FUNCTION_BLOCK FB_PID_LIMI (* PID controller with limited frame for the integrator. *)
  (* Standard: 61499-2; Description: Rather than integrating the error over all vallues, the error is integrated over the last N values. Fixed-width time intervals are required for the input. *)
  (* Version 0.0, 2017-06-15, 4DIAC-IDE, 4DIAC-Consortium *)
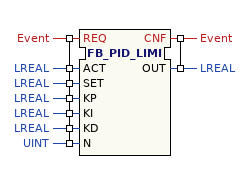
  EVENT_INPUT
    REQ WITH ACT, SET, KP, KI, KD, N; (* Normal Execution Request *)
  END_EVENT
  EVENT_OUTPUT
    CNF WITH OUT; (* Execution Confirmation *)
  END_EVENT
  VAR_INPUT
    ACT : LREAL; (* Actual value *)
    SET : LREAL; (* Set value *)
    KP : LREAL; (* Proportional coefficient *)
    KI : LREAL; (* Integral coefficient *)
    KD : LREAL; (* Derivative coefficient *)
    N : UINT := 1; (* Amount of values to look back for integral computation *)
  END_VAR
  VAR_OUTPUT
    OUT : LREAL; (* Output value = KP*(SET-ACT) + KI*INT_0_N(SET-ACT) + KD*DIFF(SET-ACT) *)
  END_VAR
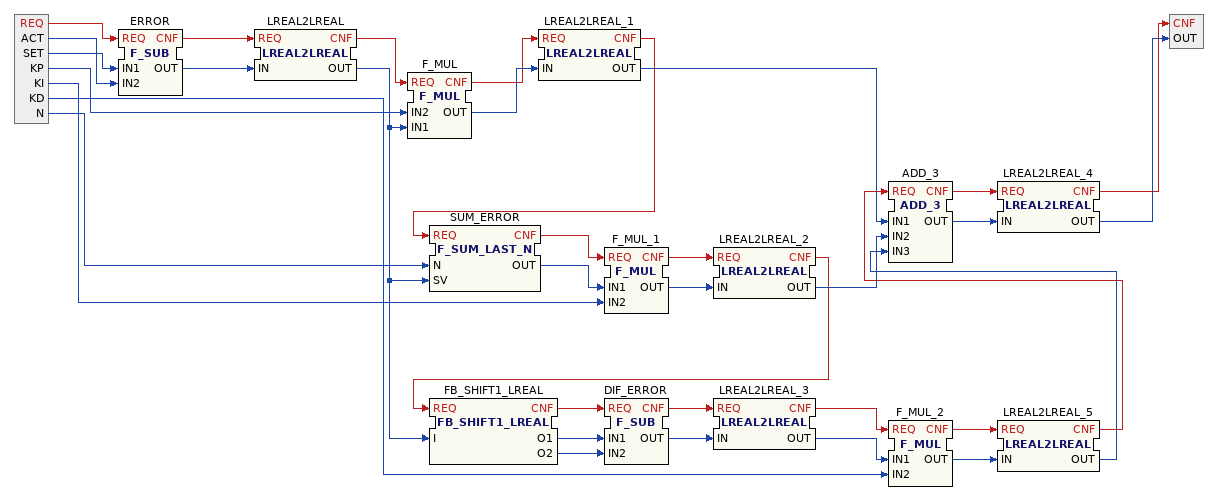
  FBS
    ERROR : F_SUB;
    SUM_ERROR : F_SUM_LAST_N;
    FB_SHIFT1_LREAL : FB_SHIFT1_LREAL;
    DIF_ERROR : F_SUB;
    F_MUL : F_MUL;
    LREAL2LREAL : LREAL2LREAL;
    LREAL2LREAL_1 : LREAL2LREAL;
    LREAL2LREAL_2 : LREAL2LREAL;
    LREAL2LREAL_3 : LREAL2LREAL;
    ADD_3 : ADD_3;
    LREAL2LREAL_4 : LREAL2LREAL;
    F_MUL_1 : F_MUL;
    F_MUL_2 : F_MUL;
    LREAL2LREAL_5 : LREAL2LREAL;
  END_FBS
  EVENT_CONNECTIONS
    REQ TO ERROR.REQ;
    FB_SHIFT1_LREAL.CNF TO DIF_ERROR.REQ;
    ERROR.CNF TO LREAL2LREAL.REQ;
    LREAL2LREAL.CNF TO F_MUL.REQ;
    F_MUL.CNF TO LREAL2LREAL_1.REQ;
    LREAL2LREAL_1.CNF TO SUM_ERROR.REQ;
    ADD_3.CNF TO LREAL2LREAL_4.REQ;
    LREAL2LREAL_4.CNF TO CNF;
    SUM_ERROR.CNF TO F_MUL_1.REQ;
    F_MUL_1.CNF TO LREAL2LREAL_2.REQ;
    DIF_ERROR.CNF TO LREAL2LREAL_3.REQ;
    LREAL2LREAL_3.CNF TO F_MUL_2.REQ;
    F_MUL_2.CNF TO LREAL2LREAL_5.REQ;
    LREAL2LREAL_5.CNF TO ADD_3.REQ;
    LREAL2LREAL_2.CNF TO FB_SHIFT1_LREAL.REQ;
  END_CONNECTIONS
  DATA_CONNECTIONS
    SET TO ERROR.IN1;
    ACT TO ERROR.IN2;
    N TO SUM_ERROR.N;
    FB_SHIFT1_LREAL.O1 TO DIF_ERROR.IN1;
    FB_SHIFT1_LREAL.O2 TO DIF_ERROR.IN2;
    KP TO F_MUL.IN2;
    ERROR.OUT TO LREAL2LREAL.IN;
    LREAL2LREAL.OUT TO F_MUL.IN1;
    F_MUL.OUT TO LREAL2LREAL_1.IN;
    LREAL2LREAL.OUT TO SUM_ERROR.SV;
    LREAL2LREAL.OUT TO FB_SHIFT1_LREAL.I;
    ADD_3.OUT TO LREAL2LREAL_4.IN;
    LREAL2LREAL_4.OUT TO OUT;
    SUM_ERROR.OUT TO F_MUL_1.IN1;
    KI TO F_MUL_1.IN2;
    F_MUL_1.OUT TO LREAL2LREAL_2.IN;
    LREAL2LREAL_1.OUT TO ADD_3.IN1;
    LREAL2LREAL_2.OUT TO ADD_3.IN2;
    DIF_ERROR.OUT TO LREAL2LREAL_3.IN;
    LREAL2LREAL_3.OUT TO F_MUL_2.IN1;
    KD TO F_MUL_2.IN2;
    F_MUL_2.OUT TO LREAL2LREAL_5.IN;
    LREAL2LREAL_5.OUT TO ADD_3.IN3;
  END_CONNECTIONS
END_FUNCTION_BLOCK
